// SIMATIC STEP 7 (V5.x) project Abdu doing magic tricks
// CPU: CPU 312C
// station: Hardware
// station: SIMATIC 300(1)
// station: P_ADR_BUS
// program: S7 Program(1)

SYMBOL_TABLE
"Debut"	I 0.0	BOOL
"Stop"	I 0.1	BOOL
"Capteur 1"	I 0.2	BOOL
"Capteur 2"	I 0.3	BOOL
"Capteur 3"	I 0.4	BOOL
"Capteur Bas"	I 1.0	BOOL
"Capteur Haut"	I 1.1	BOOL
"Capteur extrem 1"	I 1.2	BOOL
"Capteur extrem 2"	I 1.3	BOOL
"z moving"	I 1.4	BOOL
"Pret"	M 0.0	BOOL
"Reset Z"	M 0.1	BOOL
"Convoyeur"	Q 0.0	BOOL
"Convoyeur 1"	Q 0.1	BOOL
"Vert"	Q 0.2	BOOL
"Bleu"	Q 0.3	BOOL
"Gris"	Q 0.4	BOOL
"mini conv"	Q 0.5	BOOL
"Convoyeur 3"	Q 0.6	BOOL
"convoyeur 4"	Q 0.7	BOOL
"Boite Grande"	Q 1.0	BOOL
"Boite large"	Q 1.1	BOOL
"Place Axis Move"	Q 1.2	BOOL
"Mvt Z"	Q 1.3	BOOL
"Capter"	Q 1.4	BOOL
"mvt x"	Q 1.5	BOOL
"Push"	Q 1.7	BOOL
END_SYMBOL_TABLE

ORGANIZATION_BLOCK OB 1
TITLE = "Main Program Sweep (Cycle)"
VERSION : 0.1
VAR_TEMP
  OB1_EV_CLASS : BYTE ;	//Bits 0-3 = 1 (Coming event), Bits 4-7 = 1 (Event class 1)
  OB1_SCAN_1 : BYTE ;	//1 (Cold restart scan 1 of OB 1), 3 (Scan 2-n of OB 1)
  OB1_PRIORITY : BYTE ;	//Priority of OB Execution
  OB1_OB_NUMBR : BYTE ;	//1 (Organization block 1, OB1)
  OB1_RESERVED_1 : BYTE ;	//Reserved for system
  OB1_RESERVED_2 : BYTE ;	//Reserved for system
  OB1_PREV_CYCLE : INT ;	//Cycle time of previous OB1 scan (milliseconds)
  OB1_MIN_CYCLE : INT ;	//Minimum cycle time of OB1 (milliseconds)
  OB1_MAX_CYCLE : INT ;	//Maximum cycle time of OB1 (milliseconds)
  OB1_DATE_TIME : DATE_AND_TIME ;	//Date and time OB1 started
END_VAR
BEGIN
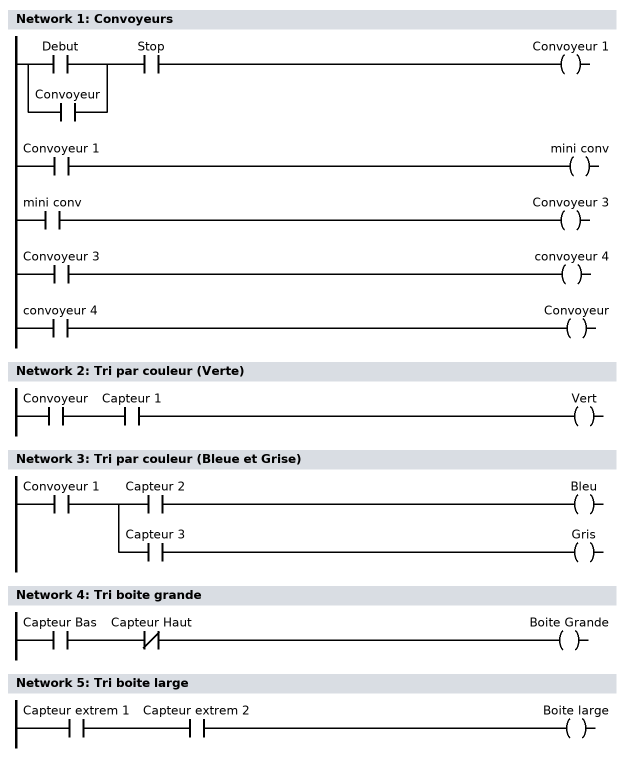
NETWORK
TITLE = Convoyeurs
      A(;
      O     "Debut";
      O     "Convoyeur";
      );
      A     "Stop";
      =     "Convoyeur 1";
      A     "Convoyeur 1";
      =     "mini conv";
      A     "mini conv";
      =     "Convoyeur 3";
      A     "Convoyeur 3";
      =     "convoyeur 4";
      A     "convoyeur 4";
      =     "Convoyeur";
NETWORK
TITLE = Tri par couleur (Verte)
      A     "Convoyeur";
      A     "Capteur 1";
      =     "Vert";
NETWORK
TITLE = Tri par couleur (Bleue et Grise)
      A     "Convoyeur 1";
      =     L 20.0;
      A     L 20.0;
      A     "Capteur 2";
      =     "Bleu";
      A     L 20.0;
      A     "Capteur 3";
      =     "Gris";
NETWORK
TITLE = Tri boite grande
      A     "Capteur Bas";
      AN    "Capteur Haut";
      =     "Boite Grande";
NETWORK
TITLE = Tri boite large
      A     "Capteur extrem 1";
      A     "Capteur extrem 2";
      =     "Boite large";
END_ORGANIZATION_BLOCK
